Universal Robots PolyScope program: wojasinski.urp

ProgramRoot setBeforeStartSequence=true; directory=/programs/USB; kinematics=(a=[0, -0.425, -0.39225, 0, 0, 0], d=[0.08916, 0, 0, 0.10915, 0.09465, 0.0823], alpha=[1.5708, 0, 0, 1.5708, -1.5708, 0], deltaTheta=[0, 0, 0, 0, 0, 0], status=notInitialized); name=wojasinski; programVersion=(project__name=PolyScope, major__version=1, minor__version=0, svn__revision=0); robotEnvironmentFileName=default; serialNumberRobot=2013210114
  BeforeStart description=COMMAND_SEQUENCE_BEFORE_PROGRAM_START; name=BeforeStart
    Assignment assignmentValueSource=0; assignmentOperatorMessage=WorkPos; expr=HomePos; operatorValueType=INTEGER; valueSource=EXPRESSION; variable=p[0, 0, 0, 0, 0, 0]
    Assignment assignmentValueSource=0; expr=WorkPos; operatorValueType=INTEGER; valueSource=EXPRESSION; variable=(name=WorkPosition, prefersPersistentValue=false, requestANewUniqueName=false)
    Assignment assignmentValueSource=0; expr=p[0,0,0,0,3.1413,0]; operatorValueType=INTEGER; valueSource=EXPRESSION; variable=(name=ObjectPos, prefersPersistentValue=false, requestANewUniqueName=false)
    Assignment assignmentValueSource=0; expr=[0,0,0,0,0,0,0]; operatorValueType=INTEGER; valueSource=EXPRESSION; variable=[0, 0, 0, 0, 0, 0, 0]
    Script type=0; expressionBranchNode=socket_open("192.168.0.110", 10000)
    Move cartesianAcceleration=1.2; cartesianSpeed=0.25; jointAcceleration=0.008726646259971648; jointSpeed=0.08726646259971647; moveAsFastAsPossible=true; sharedProcessMoveBlendRadius=0.025; featureReference=(installationNameReference=Base); motionType=PROCESS_MOVE
      Waypoint blendRadius=0.05; cartesianAcceleration=1.2; cartesianSpeed=0.25; jointAcceleration=1.3962634015954636; jointSpeed=1.0471975511965976; nextMotionTime=2.0; stoppoint=true; useSharedBlendParameter=true; useSharedParameters=true; position=TCP in base x=29.602 y=-168.865 z=522.149 mm, rx=-1.1813 ry=-1.2279 rz=1.2376 rad; joints [-269.073, -124.288, 99.982, 352.622, 178.741, 148.108] deg; positionType=VARIABLE_POSITION; variable=p[0, 0, 0, 0, 0, 0]; waypointPoseInFeatureCoordinates=(pos=(x=0.029601963106494385, y=-0.16886496724660927, z=0.5221490682021757), rot=(x=-1.1813166177317849, y=-1.2278910041760307, z=1.2375657959715258)); name=HomePos_2
  MainProgram cartesianAcceleration=1.2; cartesianSpeed=0.25; jointAcceleration=1.3962634015954636; jointSpeed=1.0471975511965976; moveAsFastAsPossible=true; sharedProcessMoveBlendRadius=0.0; featureReference=(installationNameReference=Base); motionType=JOINT_SPACE
    Script type=0; expressionBranchNode=TempPoint = socket_read_ascii_float(6)
    If expr=ExpressionVariableNode[0]==6; type=IF_NODE
      Script type=0; expressionBranchNode=ObjectPos[0] = TempPoint[1]
      Script type=0; expressionBranchNode=ObjectPos[1] = TempPoint[2]
      Script type=0; expressionBranchNode=ObjectPos[2] = TempPoint[3]
      Script type=0; expressionBranchNode=ObjectPos[3] = 0
      Script type=0; expressionBranchNode=ObjectPos[4] = 3.1413
      Script type=0; expressionBranchNode=ObjectPos[5] = 0
      Move cartesianAcceleration=0.005; cartesianSpeed=0.01; jointAcceleration=0.017453292519943295; jointSpeed=0.06981317007977318; moveAsFastAsPossible=true; sharedProcessMoveBlendRadius=0.025; featureReference=(installationNameReference=Base); motionType=JOINT_SPACE
        Waypoint blendRadius=0.05; cartesianAcceleration=1.2; cartesianSpeed=0.25; jointAcceleration=1.3962634015954636; jointSpeed=1.0471975511965976; nextMotionTime=2.0; stoppoint=true; useSharedBlendParameter=true; useSharedParameters=true; positionType=VARIABLE_POSITION; variable=(name=ObjectPos, prefersPersistentValue=false, requestANewUniqueName=false); waypointPoseInFeatureCoordinates=(pos=(x=0.0, y=0.0, z=0.0), rot=(x=0.0, y=0.0, z=0.0)); name=WorkPos_1
        Wait analogComparison=0; analogInputRange=0; analogValue=0.0; digitalValue=0; selectedAnalogSensor=-1; selectedDigitalSensor=-1; waitTime=0.5; type=TIMER_WAIT
        Waypoint blendRadius=0.05; cartesianAcceleration=1.2; cartesianSpeed=0.25; jointAcceleration=1.3962634015954636; jointSpeed=1.0471975511965976; nextMotionTime=2.0; stoppoint=true; useSharedBlendParameter=true; useSharedParameters=true; positionType=VARIABLE_POSITION; variable=(name=WorkPosition, prefersPersistentValue=false, requestANewUniqueName=false); waypointPoseInFeatureCoordinates=(pos=(x=0.0, y=0.0, z=0.0), rot=(x=0.0, y=0.0, z=0.0)); name=WorkPos_1
        Wait analogComparison=0; analogInputRange=0; analogValue=0.0; digitalValue=0; selectedAnalogSensor=-1; selectedDigitalSensor=-1; waitTime=2.0; type=TIMER_WAIT
        Waypoint blendRadius=0.05; cartesianAcceleration=1.2; cartesianSpeed=0.25; jointAcceleration=1.3962634015954636; jointSpeed=1.0471975511965976; nextMotionTime=2.0; stoppoint=true; useSharedBlendParameter=true; useSharedParameters=true; positionType=VARIABLE_POSITION; variable=p[0, 0, 0, 0, 0, 0]; waypointPoseInFeatureCoordinates=(pos=(x=0.0, y=0.0, z=0.0), rot=(x=0.0, y=0.0, z=0.0)); name=HomePos_1
      Script type=0; expressionBranchNode=socket_send_string("OK")
